// TIA Portal V16 export
// export: Created 2021-07-12T14:47:18.0432485Z, ExportSetting WithDefaults, DisplayName Totally Integrated Automation Portal, DisplayVersion V16, DisplayName TIA Portal Version Control Interface, DisplayVersion V16, DisplayName TIA Portal Openness, DisplayVersion V16, DisplayName STEP 7 Professional, DisplayVersion V16, DisplayName STEP 7 Safety, DisplayVersion V16, DisplayName WinCC Professional, DisplayVersion V16
TYPE "SimaHydTO_typeAxesArrayVCharMeasurement"
TITLE = SimaHydTO_typeAxesArrayVCharMeasurement
// Axis array of HMI axis selection
// stored: IsFailsafeCompliant false
   STRUCT
      requestForward { ExternalAccessible := 'False'; ExternalVisible := 'False'; ExternalWritable := 'False'} : Bool;   // Switches the digital valves to move in the positive direction
      requestBackward { ExternalAccessible := 'False'; ExternalVisible := 'False'; ExternalWritable := 'False'} : Bool;   // Switches the digital valves to move in the negative direction
      enableRampingForward { ExternalAccessible := 'False'; ExternalVisible := 'False'; ExternalWritable := 'False'} : Bool := True;   // Enable ramping of Q-Output value (voltage) in positivedirection
      enableRampingBackward { ExternalAccessible := 'False'; ExternalVisible := 'False'; ExternalWritable := 'False'} : Bool := True;   // Enable ramping of Q-Output value (voltage) in negative direction
   END_STRUCT;
END_TYPE
